# B&R Automation Studio project LiquidControlOfTank
Automation Studio 4.3.7.46 SP

## Configuration Config1

CPU 4PP065.0571-X74, AutomationRuntime E4.34, Build 4.1.2, Vc V4.34.1

### Task classes (Cpu.sw)
```
Cyclic#4:
  Master <- Modbus.Master.prg
  Visu_1 <- Visualisation.Visu_1.prg
DataObjects: datamod <- Modbus.datamod.dob
VcDataObjects: Visu1 <- Visualisation.Visu1.dob
Binaries: udbdef, vcrt, vccnum, vcctext, Visu101, vcpfmtcx, Visu103, Visu102, vcfile, vcgclass, vcpdsw, vccshape, arial, vccbmp, vcmgr, vcchspot, vcdsloc, vcfntttf, vccovl, vcshared, arialbd, vcalarm, vcptelo, vccdt, vccbtn, vcbclass, vcpfpp30, vcdsint, vctcal, TCData, vcpdpp30, vccalarm, vccbar, arconfig, User, ashwd, sysconf, ashwac, Role, asfw, iomap
Libraries: asstring, AsBrStr, DRV_mbus, DataObj, runtime, become, dvframe, vcresman, fileio, asieccon
```

### Hardware
```
4PP065_0571_X74 : 4PP065.0571-X74 v1.1.5.0
  Connector IF5:
    ActivateDevice = 1
    Mode = Manual
    InternetAddress = 192.168.1.10
    SubnetMask = 255.255.255.0
  ConfigurationID = 01082018_Config1
  TimeZone = 260
  VcObjectName = Visu1
4PP065_IF23-1 : 4PP065.IF23-1 v1.0.4.0  [SS -> 4PP065_0571_X74.SS1]
  Connector IF1:
    Baudrate = 19200
    Parity = N
```

## Configuration Config2

CPU X20cCP1301, AutomationRuntime E4.34, Build 4.1.2, Vc V4.34.1

### Task classes (Cpu.sw)
```
Cyclic#4:
  Program1 <- Program1.prg
  Visu_1 <- Visu_1.prg
VcDataObjects: Visu1 <- Visu1.dob
Binaries: vcfile, vcrt, vcfntttf, vcctext, arial, vccdt, vcmgr, vcpkat, vccovl, vccnum, vcpfar00, vcdsint, vcpdvnc, vcshared, Visu102, vcpdsw, vcalarm, vcchspot, vccbtn, Visu101, vcgclass, vcdsloc, arialbd, vcnet, TCData, vctcal, udbdef, Visu103, vcbclass, vccshape, vccbmp, ashwac, User, ashwd, arconfig, sysconf, Role, asfw, iomap
Libraries: become, standard, fileio, dataobj, vcresman, runtime
```

### Hardware
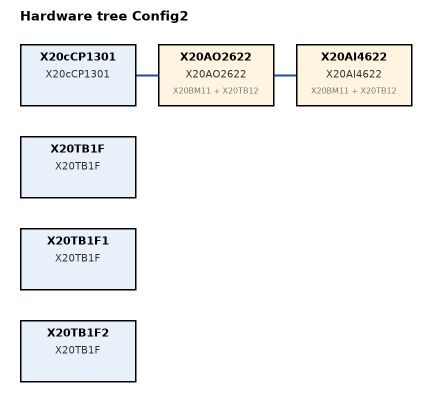
```
X20AI4622 : X20AI4622 v1.0.4.0  [SS1 -> X20TB12a.SS; SL -> X20BM11a.SL1]
  LowerLimit = 0
  ChannelType01 = 4 to 20mA
  ChannelType02 = 4 to 20mA
X20AO2622 : X20AO2622 v1.1.0.0  [SS1 -> X20TB12.SS; SL -> X20BM11.SL1]
  ChannelType01 = 4 to 20mA
  ChannelType02 = 4 to 20mA
X20BM11 : X20BM11 v1.0.0.1  [X2X1 -> X20cCP1301.IF6]
X20BM11a : X20BM11 v1.0.0.1  [X2X1 -> X20BM11.X2X2]
X20TB12 : X20TB12 v1.0.0.0
X20TB12a : X20TB12 v1.0.0.0
X20TB1F : X20TB1F v1.0.0.0
X20TB1F1 : X20TB1F v1.0.0.0
X20TB1F2 : X20TB1F v1.0.0.0
X20cCP1301 : X20cCP1301 v1.3.2.0  [X1 -> X1.SL; X2 -> X2.SL; X3 -> X3.SL]
  Module X1 (Type=X1, Virtual=true, Version=1.3.2.0)
    Connection (Connector=SS1, TargetModule=X20TB1F, TargetConnector=SS)
    Connection (Connector=SL, TargetModule=X20cCP1301, TargetConnector=X1)
  Module X2 (Type=X2, Virtual=true, Version=1.3.2.0)
    Connection (Connector=SS1, TargetModule=X20TB1F1, TargetConnector=SS)
    Connection (Connector=SL, TargetModule=X20cCP1301, TargetConnector=X2)
  Module X3 (Type=X3, Virtual=true, Version=1.3.2.0)
    Connection (Connector=SS1, TargetModule=X20TB1F2, TargetConnector=SS)
    Connection (Connector=SL, TargetModule=X20cCP1301, TargetConnector=X3)
  Connector IF2:
    ActivateDevice = 1
    Mode = Manual
    InternetAddress = 192.168.0.10
    SubnetMask = 255.255.255.0
    Vnc1
    VncVcObjectName1 = Visu1
    VncKeyMappingFile1 = VC\PS2-Keyboard.dis
    VncRefreshRate1 = 100
  ConfigurationID = 01082018_Config2
```

### IoMap.iom - X20cCP1301/IoMap.iom
```iecst
VAR_CONFIG
	::VALVE.feedback.raw AT %IW."X20AI4622".AnalogInput01;
	::TANK.level.raw AT %IW."X20AI4622".AnalogInput02;
	Cyclic#1.::ai_input_status AT %IB."X20AI4622".StatusInput01;
	::PUMP.status_running AT %IX."X2".DigitalInput01;
	::PUMP.status_remote AT %IX."X2".DigitalInput02;
	::VALVE.status_remote AT %IX."X2".DigitalInput03;
	::VALVE.status_local AT %IX."X2".DigitalInput04;
	::VALVE.button_open AT %IX."X2".DigitalInput05;
	::VALVE.button_close AT %IX."X2".DigitalInput06;
	::VALVE.button_stop AT %IX."X2".DigitalInput07;
	::PUMP.cmd_on AT %IX."X3".StatusDigitalOutput01;
	::VALVE.signal_valve_opened AT %IX."X3".StatusDigitalOutput02;
	::VALVE.signal_valve_closed AT %IX."X3".StatusDigitalOutput03;
	::VALVE.cmd_valve_open AT %IX."X3".StatusDigitalOutput04;
	::VALVE.cmd_valve_close AT %IX."X3".StatusDigitalOutput05;
END_VAR
```

## Configuration Config3

CPU X20CP1301, AutomationRuntime E4.34, Build 4.1.2, Vc V4.34.1

### Task classes (Cpu.sw)
```
Cyclic#4:
  Visu_1 <- Visualisation.Visu_1.prg
  Main_Progr <- Main_Program.prg
  Slave <- Modbus.Slave.prg
DataObjects: datamod <- Modbus.datamod.dob
VcDataObjects: Visu1 <- Visualisation.Visu1.dob
Binaries: Visu101, vccbar, vcrt, vcfntttf, vcctext, arial, vccdt, vcmgr, vcpkat, vccovl, vcchspot, vcdsint, vcpfx20, vcpdvnc, vcshared, Visu102, vcpdsw, vcfile, vcalarm, vccbtn, vccnum, vcgclass, vcdsloc, arialbd, vcnet, TCData, vctcal, udbdef, vccalarm, Visu103, vcbclass, vccshape, vccbmp, ashwac, User, ashwd, arconfig, sysconf, Role, asfw, iomap, vcpfar00
Libraries: become, vcresman, fileio, dataobj, ashw, runtime, standard, asstring, drv_mbus, dvframe
```

### Hardware
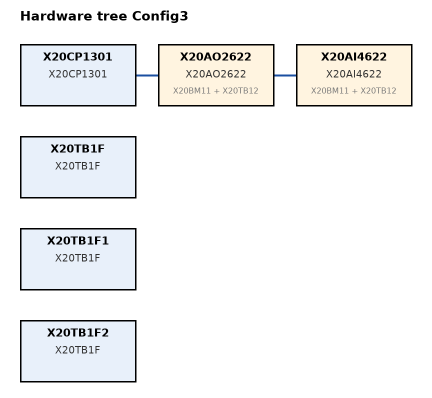
```
X20AI4622 : X20AI4622 v1.0.4.0  [SS1 -> X20TB12.SS; SL -> X20BM11.SL1]
  LowerLimit = 0
  ChannelType01 = 4 to 20mA
  ChannelType02 = 4 to 20mA
  ChannelType03 = 4 to 20mA
  ChannelType04 = 4 to 20mA
X20AO2622 : X20AO2622 v1.1.0.0  [SS1 -> X20TB12a.SS; SL -> X20BM11a.SL1]
  ChannelType01 = 4 to 20mA
  ChannelType02 = 4 to 20mA
X20BM11 : X20BM11 v1.0.0.1  [X2X1 -> X20BM11a.X2X2]
X20BM11a : X20BM11 v1.0.0.1  [X2X1 -> X20CP1301.IF6]
X20CP1301 : X20CP1301 v1.3.2.0  [X1 -> X1.SL; X2 -> X2.SL; X3 -> X3.SL]
  Module X1 (Type=X1, Virtual=true, Version=1.3.2.0)
    Connection (Connector=SS1, TargetModule=X20TB1F, TargetConnector=SS)
    Connection (Connector=SL, TargetModule=X20CP1301, TargetConnector=X1)
  Module X2 (Type=X2, Virtual=true, Version=1.3.2.0)
    Connection (Connector=SS1, TargetModule=X20TB1F1, TargetConnector=SS)
    Connection (Connector=SL, TargetModule=X20CP1301, TargetConnector=X2)
  Module X3 (Type=X3, Virtual=true, Version=1.3.2.0)
    Connection (Connector=SS1, TargetModule=X20TB1F2, TargetConnector=SS)
    Connection (Connector=SL, TargetModule=X20CP1301, TargetConnector=X3)
  Connector IF1:
    Baudrate = 19200
    Parity = N
  Connector IF2:
    ActivateDevice = 1
    Mode = Manual
    InternetAddress = 192.168.1.100
    SubnetMask = 255.255.255.0
    Vnc1
    VncVcObjectName1 = Visu1
    VncKeyMappingFile1 = VC\PS2-Keyboard.dis
    VncRefreshRate1 = 100
  ConfigurationID = LiquidControlOfTank_Config3
X20TB12 : X20TB12 v1.0.0.0
X20TB12a : X20TB12 v1.0.0.0
X20TB1F : X20TB1F v1.0.0.0
X20TB1F1 : X20TB1F v1.0.0.0
X20TB1F2 : X20TB1F v1.0.0.0
```

### IoMap.iom - X20CP1301/IoMap.iom
```iecst
VAR_CONFIG
	::VALVE.feedback.raw AT %IW."X20AI4622".AnalogInput01;
	::TANK.level.raw AT %IW."X20AI4622".AnalogInput02;
	::PUMP.status_running AT %IX."X2".DigitalInput01;
	::PUMP.status_remote AT %IX."X2".DigitalInput02;
	::VALVE.status_remote AT %IX."X2".DigitalInput03;
	::VALVE.status_local AT %IX."X2".DigitalInput04;
	::VALVE.button_open AT %IX."X2".DigitalInput05;
	::VALVE.button_close AT %IX."X2".DigitalInput06;
	::VALVE.button_stop AT %IX."X2".DigitalInput07;
	::PUMP.cmd_on AT %QX."X3".DigitalOutput01;
	::VALVE.signal_valve_opened AT %QX."X3".DigitalOutput02;
	::VALVE.signal_valve_closed AT %QX."X3".DigitalOutput03;
	::VALVE.cmd_valve_open AT %QX."X3".DigitalOutput04;
	::VALVE.cmd_valve_close AT %QX."X3".DigitalOutput05;
END_VAR
```

## Logical view

Binary libraries used (declarations not repeated): operator, runtime, astime, AsIecCon, asstring, AsBrStr, DRV_mbus, DataObj, standard, dvframe

### Global.typ - Global data types
```iecst
TYPE
	Pump_typ : 	STRUCT
		status_running : BOOL; (*Статус насоса "Включен / Выключен"*)
		status_remote : BOOL; (*Статус переключателя "Дистанционный"*)
		cmd_on : BOOL; (*Команда "Включить" насос*)
		button_stop : BOOL; (*Кнопка "Стоп"*)
	END_STRUCT;
	Valve_typ : 	STRUCT
		status_remote : BOOL; (*Статус переключателя "Дистанционный"*)
		status_local : BOOL; (*Статус переключателя "Местный"*)
		button_open : BOOL; (*Кнопка "Открыть" задвижку*)
		button_close : BOOL; (*Кнопка "Закрыть" задвижку*)
		button_stop : BOOL; (*Кнопка "Стоп" задвижку*)
		signal_valve_opened : BOOL; (*Сигнал на индикацию "Задвижка открыта"*)
		signal_valve_closed : BOOL; (*Сигнал на индикацию "Задвижка закрыта"*)
		cmd_valve_open : BOOL; (*Команда открыть задвижку*)
		cmd_valve_close : BOOL; (*Команда закрыть задвижку*)
		feedback : Analog_FB; (*Состояние задвижки (0-100%)*)
	END_STRUCT;
	Tank_typ : 	STRUCT
		level : Analog_FB; (*Уровень жидкости в резервуаре*)
	END_STRUCT;
END_TYPE
```

### Global.var - Global variables
```iecst
(*Задвижка*)
VAR
	VALVE : Valve_typ;
END_VAR
(*Насос*)
VAR
	PUMP : Pump_typ;
END_VAR
(*Резервуар*)
VAR
	TANK : Tank_typ;
END_VAR
(*Аналоговые сигналы*)
VAR
	ai_input_status : USINT; (*Состояние аналоговых каналов*)
END_VAR
(*Примеры для аларма*)
VAR
	alarm : ARRAY[0..19] OF BOOL;
	general_alarm : BOOL;
END_VAR
(*Insert your comment here.*)
VAR
	timer_for_valve : UINT; (*Таймер для открытия задвижки *)
	level_limits : Analog_Limits_typ; (*Технологические значения диапазонов уровня в резервуаре*)
	cmd_pump_on : BOOL; (*Команда для запуска насоса в дистанционном режиме*)
	cmd_pump_off : BOOL; (*Команда для останова насоса в дистанционном режиме*)
	cmd_valve_open : BOOL; (*Команда для открытия задвижки в дистанционном режиме*)
	cmd_valve_close : BOOL; (*Команда для закрытия задвижки в дистанционном режиме*)
	cmd_valve_stop : BOOL; (*Команда для останова задвижки в дистанционном режиме*)
	mode_remote_auto : BOOL; (*Режим дистанционный "Автомат"*)
	mode_remote_manual : BOOL; (*Режим дистанционный "Ручной"*)
	block_auto : BOOL; (*Блокировка кнопки "Автомат" на Touch - панели*)
	block_manual : BOOL; (*Блокировка кнопки "Manual" на Touch - панели*)
	block_valve_cmd : BOOL; (*Блокировка кнопок управления задвижкой в режиме "Дистанционный"*)
	block_pump_cmd : BOOL; (*Блокировка кнопок управления насосом в режиме "Дистанционный"*)
	ack_alarms : BOOL;
END_VAR
```

### Package Logical/Libraries - Global libraries

### Library Logical/Libraries/become (ANSIC, version 1.00.0)

#### Types.typ - Exported data types
```iecst
(*Аналоговый сигнал*)

TYPE
	Analog_Settings_type : 	STRUCT
		scale_h : REAL;
		scale_l : REAL;
		offset : REAL;
	END_STRUCT;
	Analog_Limits_typ : 	STRUCT
		HiHi : REAL;
		Hi : REAL;
		Lo : REAL;
		LoLo : REAL;
		hys : REAL;
	END_STRUCT;
	anaAlarmsEnum :
		(
		SIGNAL_NO_ALARM := 0,
		SIGNAL_OVER := 1,
		SIGNAL_UNDER := 2,
		SIGNAL_OPEN_LINE := 4,
		SIGNAL_HI_HI := 8,
		SIGNAL_HI := 16,
		SIGNAL_LO := 32,
		SIGNAL_LO_LO := 64
		);
END_TYPE

(*Общие*)

TYPE
	localRemoteSwitchEnum :
		( (*Положение ключа управления*)
		SW_OFF := 0,
		SW_LOCAL := 1,
		SW_REMOTE := 2
		);
END_TYPE
```

#### become.fun - Exported functions and function blocks
```iecst
FUNCTION_BLOCK Analog_FB (*Аналоговый сигнал*)
	VAR_INPUT
		raw : INT; (*"сырое" значение с модуля*)
		ai_input_status : BYTE; (*байт-статус с модуля*)
		ai_channel_num : BYTE; (*номер аналогового входа*)
	END_VAR
	VAR_OUTPUT
		value : REAL; (*смасштабированное значение в физических единицах*)
	END_VAR
	VAR
		sett : Analog_Settings_type;
		limits : Analog_Limits_typ;
		alarms : anaAlarmsEnum;
	END_VAR
	VAR_INPUT
		adc_up : INT; (*Верхняя шкала*)
		adc_dn : INT; (*Нижняя шкала*)
	END_VAR
END_FUNCTION_BLOCK
```

#### Analog.c
```c
#include <bur/plctypes.h>
#include "become.h"

void Analog_FB (struct Analog_FB* inst)
{
	INT adc_up = inst->adc_up;
	INT adc_dn = inst->adc_dn;
	REAL raw, phys;
	BOOL signal_fail;
	BYTE status, channel_number;
	anaAlarmsEnum tAlarms = 0;

	/* Диагностика состояния аналогового сигнала*/
	/* Нумерация каналов начинается с 0, поэтому "номер канала" - 1.
	   Статусы каналов разбиты на 2 переменные, поэтому каналы 5-8
	   заново начинаюся с 0, но во второй переменной */

	channel_number = inst->ai_channel_num >4 ? inst->ai_channel_num - 5 : inst->ai_channel_num - 1;

	status = (inst->ai_input_status >> (channel_number << 1)) & 0x03;

	switch (status)
	{
		case 0x01:
			/* Lower limit */
			tAlarms |= SIGNAL_UNDER;
			//raw = inst->sett.scale_l;
			break;
		case 0x02:
			/* Upper limit */
			tAlarms |= SIGNAL_OVER;
			//raw = inst->sett.scale_h;
			break;
		case 0x03:
			/* Обрыв */
			tAlarms |= SIGNAL_OPEN_LINE;
			//raw = inst->sett.scale_l;
			break;
		default:
			//raw = inst->sett.invert_input_scale ? (32767 - inst->raw) : inst->raw;
			raw = inst->raw;
			//tAlarms = signal_no_alarm;
			break;
	}

	signal_fail = (tAlarms != 0);

	/* Представление сигнала в инженерных единицах */
	phys = (raw - adc_dn)*(inst->sett.scale_h - inst->sett.scale_l)/(adc_up - adc_dn) + inst->sett.scale_l + inst->sett.offset;

	inst->alarms = (inst->alarms & ~(SIGNAL_UNDER | SIGNAL_OVER | SIGNAL_OPEN_LINE)) | tAlarms;

	if ((!signal_fail) && (phys >= inst->limits.HiHi))
		inst->alarms |= SIGNAL_HI_HI;
	if ((signal_fail) || (phys < inst->limits.HiHi - inst->limits.hys))
		inst->alarms &= ~SIGNAL_HI_HI;

	if ((!signal_fail) && (phys >= inst->limits.Hi))
		inst->alarms |= SIGNAL_HI;
	if ((signal_fail) || (phys < inst->limits.Hi - inst->limits.hys))
		inst->alarms &= ~SIGNAL_HI;

	if ((!signal_fail) && (phys <= inst->limits.Lo))
		inst->alarms |= SIGNAL_LO;
	if ((signal_fail) || (phys > inst->limits.Lo + inst->limits.hys))
		inst->alarms &= ~SIGNAL_LO;

	if ((!signal_fail) && (phys <= inst->limits.LoLo))
		inst->alarms |= SIGNAL_LO_LO;
	if ((signal_fail) || (phys > inst->limits.LoLo + inst->limits.hys))
		inst->alarms &= ~SIGNAL_LO_LO;

	inst->value = phys;
}
```

### Program Logical/Main_Program (ANSIC)

#### Variables.var
```iecst
VAR
	timer_for_pump : USINT; (*Таймер для запуска насоса*)
	TON_valve : TON; (*Таймер для открытия/закрытия задвижки*)
	TON_pump : TON; (*Таймер для старта/останова насоса*)
	virtual_valve_close : BOOL; (*Самоподхват для кнопки  останова насоса*)
	virtual_valve_open : BOOL; (*Самоподхват для кнопки запуска насоса*)
END_VAR
```

#### Cyclic.c
```c
#include <bur/plc.h>
#include <bur/plctypes.h>
#include <standard.h>
#include <become.h>

#ifdef _DEFAULT_INCLUDES
#include <AsDefault.h>
#endif

_LOCAL BOOL pump_status_changed, pump_prev_status;

/* 	alarm[0] - Авария запуска насоса;
	alarm[1] - Авария открытия задвижки;
	alarm[2] - Авария выключения насоса;
	alarm[3] - Авария закрытия задвижки;
	alarm[4] - Сработала кнопка останова задвижки;
	alarm[5] - Верхний уровень в резервуаре;
	alarm[6] - Нижний уровень в резервуаре;
	alarm[7] - Сработала кнопка останова насоса*/

BOOL TimerValve_func(BOOL start, INT presetTime){

	/* Таймер умножаем на 1000 (равно 1 секунде) */
	TON_valve.IN = start;
	TON_valve.PT = presetTime * 1000;
	TON(&TON_valve);

	return TON_valve.Q;
}

BOOL TimerPump_func(BOOL start, INT presetTime){

	/* Таймер умножаем на 1000 (равно 1 секунде) */
	TON_pump.IN = start;
	TON_pump.PT = presetTime * 1000;
	TON(&TON_pump);

	return TON_pump.Q;
}

void Alarm_func(){

	/* Вержний уровень в резервуаре */
	if (TANK.level.value >= TANK.level.limits.HiHi){
		alarm[5] = 1;
		alarm[6] = 0;
	}
	/* Нижний уровень в резервуаре */
	if(TANK.level.value <= TANK.level.limits.LoLo){
		alarm[6] = 1;
		alarm[5] = 0;
	}
	/* Если уровень в пределах нормы, то сбросить алармы по уровню */
	if ((TANK.level.value > TANK.level.limits.LoLo) && (TANK.level.value < TANK.level.limits.HiHi)){
		alarm[5] = 0;
		alarm[6] = 0;
	}
	if (alarm[0] || alarm[7] || alarm[2]){
		PUMP.cmd_on = 0;
	}
	if (alarm[0]){
		cmd_pump_on = 0;
	}
	if (alarm[2]) {
		cmd_pump_off = 0;
	}
	if (alarm[1] || alarm[4]){
		VALVE.cmd_valve_open = 0;
		cmd_valve_open = 0;
	}
	if (alarm[3] || alarm[4]){
		VALVE.cmd_valve_close = 0;
		cmd_valve_close = 0;
	}
	if (alarm[0] || alarm[1] || alarm[2] || alarm[3]){
		mode_remote_manual = 0;
	}
	if (alarm[0] || alarm[1] || alarm[2] || alarm[3] || alarm[4] || alarm[7]){
		mode_remote_auto = 0;}
}

void _CYCLIC ProgramCyclic(void){

	Alarm_func();
	/* =========================== */
	VALVE.feedback.adc_up = 32767;
	VALVE.feedback.adc_dn = 0;
	Analog_FB(&VALVE.feedback);
	/* =========================== */
	TANK.level.adc_up = 11000;
	TANK.level.adc_dn = 0;
	Analog_FB(&TANK.level);

	/* Мониторинг состояния задвижки */
	VALVE.signal_valve_opened = (VALVE.feedback.value == 100) ? 1 : 0;
	VALVE.signal_valve_closed = (VALVE.feedback.value == 0) ? 1 : 0;

	/* Если насос и задвижка в дистанционном режиме, то разрешение на их запуск с панели" */
	if (PUMP.status_remote || VALVE.status_remote){

		/* При нажатии кнопки "Стоп" запустить триггер */
		if (!VALVE.button_stop){
			mode_remote_auto = 0;
			mode_remote_manual = 0;
			VALVE.cmd_valve_close = 0;
			VALVE.cmd_valve_open = 0;
			cmd_valve_close = 0;
			cmd_valve_open = 0;
			TimerPump_func(0, 0);
			TimerValve_func(0, 0);
			alarm[4] = 1; // Сработала кнопка останова задвижки
		}

		pump_status_changed = PUMP.status_running ^ pump_prev_status;	// Status is changed
		pump_prev_status = PUMP.status_running;						 	// Previous status of pump

		/* При нажатии на кнопку "Стоп" по месту, насос должен остановиться, выйти из всех режимов и обнулить команды */
		if (PUMP.cmd_on && pump_status_changed && (pump_prev_status == 0)){
			PUMP.cmd_on = 0;
			mode_remote_auto = 0;
			mode_remote_manual = 0;
			cmd_pump_on = 0;
			cmd_pump_off = 0;
			alarm[7] = 1;
		}

		/* Если на панели выбран режим "Автомат" */
		if (mode_remote_auto){

			/* Открытие задвижки и включение насоса по достижению верхней уставки */
			if (TANK.level.value >= level_limits.Hi){
				VALVE.cmd_valve_close = 0;
				VALVE.cmd_valve_open = 1;

				/* Если задвижка открылась подаем сигнал на останов насоса */
				if (VALVE.feedback.value == 100){
					TimerValve_func(0, 0);
					VALVE.cmd_valve_open = 0;
					VALVE.signal_valve_opened = 1;
					PUMP.cmd_on = 1;
					alarm[1] = 0;

					/* Насос выключился */
					if (PUMP.status_running){
						TimerPump_func(0, 0);
						alarm[0] = 0;
					}

					/* Если насос не включился */
					if (!PUMP.status_running){
						if (TimerPump_func(1, timer_for_pump)){
							PUMP.cmd_on = 0;
							TimerPump_func(0, 0);
							mode_remote_auto = 0;
							MB0[14] = mode_remote_auto;
							alarm[0] = 1;
						}
					}
				}
				if (VALVE.feedback.value < 100){  /* В течение заданного времени задвижка не открылась*/
					if (TimerValve_func(1, timer_for_valve)){
						VALVE.cmd_valve_open = 0;
						TimerValve_func(0, 0);
						mode_remote_auto = 0;
						MB0[14] = mode_remote_auto;
						alarm[1] = 1;
					}
				}
			}

			/* Закрытие задвижки и выключение насоса по достижению нижней уставки */
			if (TANK.level.value <= level_limits.Lo){
				PUMP.cmd_on = 0;

				/* Насос выключен - сигнал на закрытие задвижки */
				if (!PUMP.status_running){
					VALVE.cmd_valve_open = 0;
					VALVE.cmd_valve_close = 1;
					TimerPump_func(0, 0);
					alarm[2] = 0;

					/* Если задвижка закрылась */
					if (VALVE.feedback.value == 0){
						VALVE.cmd_valve_close = 0;
						VALVE.signal_valve_closed = 1;
						TimerValve_func(0, 0);
						alarm[3] = 0;
					}

					/* Если сработал таймер и задвижка не закрылась */
					if (VALVE.feedback.value > 0){
						if (TimerValve_func(1, timer_for_valve)){
							VALVE.cmd_valve_close = 0;
							VALVE.cmd_valve_open = 0;
							TimerValve_func(0, 0);
							mode_remote_auto = 0;
							MB0[14] = mode_remote_auto;
							alarm[3] = 1;
						}
					}
				}

				/* Если насос не выключился, то-  */
				if (PUMP.status_running){
					if (TimerPump_func(1, timer_for_pump)){
						PUMP.cmd_on = 0;
						TimerPump_func(0, 0);
						mode_remote_auto = 0;
						MB0[14] = mode_remote_auto;
						alarm[2] = 1;
					}
				}
			}
		}

		/* Если на панели выбран режим "Manual" */
		if (mode_remote_manual){

			/* Open valve from Touch panel */
			if (cmd_valve_open){
				VALVE.cmd_valve_close = 0;
				VALVE.cmd_valve_open = 1;

				/* Задаем таймер на открытие задвижки */
				if (VALVE.feedback.value == 100){
					TimerValve_func(0, 0);
					VALVE.cmd_valve_open = 0;
					cmd_valve_open = 0;
					MB0[16] = cmd_valve_open;				// [16] Coil
					VALVE.signal_valve_opened = 1;
					alarm[1] = 0;
				}
				if (VALVE.feedback.value < 100){
					if (TimerValve_func(1, timer_for_valve)){
						VALVE.cmd_valve_open = 0;
						cmd_valve_open = 0;
						MB0[16] = cmd_valve_open;				// [16] Coil
						TimerValve_func(0, 0);
						mode_remote_manual = 0;
						MB0[15] = mode_remote_manual;
						alarm[1] = 1;
					}
				}
			}

			/* Close valve from Touch panel */
			if (cmd_valve_close){
				VALVE.cmd_valve_open = 0;
				VALVE.cmd_valve_close = 1;

				/* Задаем таймер на закрытие задвижки */
				if (VALVE.feedback.value == 0){
					TimerValve_func(0, 0);
					VALVE.cmd_valve_close = 0;
					VALVE.signal_valve_closed = 1;
					cmd_valve_close = 0;
					MB0[17] = cmd_valve_close;				// [17] Coil
					alarm[3] = 0;
				}
				if (VALVE.feedback.value > 0) {
					if(TimerValve_func(1, timer_for_valve)){
						VALVE.cmd_valve_close = 0;
						cmd_valve_close = 0;
						MB0[17] = cmd_valve_close;
						TimerValve_func(0, 0);
						mode_remote_manual = 0;
						MB0[15] = mode_remote_manual;
						alarm[3] = 1;
					}
				}
			}

			/* Turn pump on from Touch panel */
			if (cmd_pump_on){
				PUMP.cmd_on = 1;

				if(PUMP.status_running){
					TimerPump_func(0, 0);
					cmd_pump_on = 0;
					MB0[19] = cmd_pump_on;					// [19] Coil
					alarm[0] = 0;
				}

				/*Если сработал таймер и насос не включился */
				if (!PUMP.status_running){
					if (TimerPump_func(1, timer_for_pump)){
						PUMP.cmd_on = 0;
						cmd_pump_on = 0;
						MB0[19] = cmd_pump_on;					// [19] Coil
						TimerPump_func(0, 0);
						mode_remote_manual = 0;
						MB0[15] = mode_remote_manual;
						alarm[0] = 1;
				}
				}
			}

			/* Turn pump off from Touch panel */
			if (cmd_pump_off){
				PUMP.cmd_on = 0;

				if (!PUMP.status_running){
					TimerPump_func(0, 0);
					cmd_pump_off = 0;
					MB0[20] = cmd_pump_off;					// [20] Coil
					alarm[2] = 0;
				}

				/* Если сработал таймер и насос не выключился (залип пускатель и т.п) */
				if (PUMP.status_running){
					if (TimerPump_func(1, timer_for_pump)){
						PUMP.cmd_on = 0;
						cmd_pump_off = 0;
						MB0[20] = cmd_pump_off;
						TimerPump_func(0, 0);
						mode_remote_manual = 0;
						MB0[15] = mode_remote_manual;
						alarm[2] = 1;
					}
				}
			}

			/* Stop valve from Touch panel */
			if (cmd_valve_stop){
				VALVE.cmd_valve_close = 0;
				VALVE.cmd_valve_open = 0;
				cmd_valve_close = 0;
				cmd_valve_open = 0;
				cmd_valve_stop = 0;
				MB0[18] = cmd_valve_stop;				// [18] Coil
				TimerValve_func (0, 0);
			}
		}
	}

	/* Если переключатель режима насоса не в дистанционном */
	if (!PUMP.status_remote)
		PUMP.cmd_on = 0;

	/* Если переключатель режима задвижки в положении "0" */
	if (!VALVE.status_local && !VALVE.status_remote){
		VALVE.cmd_valve_open = 0;
		VALVE.cmd_valve_close = 0;
		cmd_valve_close = 0;
		cmd_valve_open = 0;
		mode_remote_auto = 0;
		TimerValve_func(0, 0);
		virtual_valve_close = 0;
		virtual_valve_open = 0;
	}

	/* Если переключатель режима задвижки в "Местное"*/
	if (VALVE.status_local){

		//mode_remote_auto = 0;
		//cmd_valve_close = 0;
		//cmd_valve_open = 0;

		/* Если по месту нажаната кнопка "Открыть" */
		if (VALVE.button_open || virtual_valve_open){
			virtual_valve_open = 1;
			VALVE.cmd_valve_close = 0;
			VALVE.cmd_valve_open = 1;

			/* Если сработал таймер и задвижка открылась */
			if (VALVE.feedback.value == 100){
				VALVE.signal_valve_opened = 1;
				VALVE.cmd_valve_open = 0;
				virtual_valve_open = 0;
				TimerValve_func(0, 0);
				alarm[1] = 0;
			}

			 /* В течение заданного времени задвижка не открылась*/
			if (VALVE.feedback.value < 100){
				if (TimerValve_func(1, timer_for_valve)){
					TimerValve_func(0, 0);
					VALVE.cmd_valve_open = 0;
					virtual_valve_open = 0;
					alarm[1] = 1;
				}
			}
		}

		/* Если по месту нажаната кнопка "Закрыть" */
		if (VALVE.button_close || virtual_valve_close){
			virtual_valve_close = 1;
			VALVE.cmd_valve_open = 0;
			VALVE.cmd_valve_close = 1;

			/* Если сработал таймер и задвижка не закрылась */
			if (VALVE.feedback.value == 0){
				VALVE.signal_valve_closed = 1;
				VALVE.cmd_valve_close = 0;
				virtual_valve_close = 0;
				TimerValve_func(0, 0);
				alarm[3] = 0;
			}
			if (TimerValve_func(1, timer_for_valve) && (VALVE.feedback.value > 0)){
				TimerValve_func(0, 0);
				VALVE.cmd_valve_close = 0;
				virtual_valve_close = 0;
				alarm[3] = 1;
			}
		}

		/* Если по месту нажаната кнопка "Стоп" */
		if(!VALVE.button_stop){
			VALVE.cmd_valve_close = 0;
			VALVE.cmd_valve_open = 0;
			TimerPump_func(0,0);
			TimerValve_func(0, 0);
			virtual_valve_close = 0;
			virtual_valve_open = 0;
			alarm[4] = 1; 						// Кнопка "Стоп" по месту
		}

	}
}
```

#### Init.c
```c
#include <bur/plctypes.h>

#ifdef _DEFAULT_INCLUDES
	#include <AsDefault.h>
#endif

void _INIT ProgramInit(void)
{
	VALVE.feedback.sett.scale_h = 100;
	VALVE.feedback.sett.scale_l = 0;
	timer_for_valve = 60;

	TANK.level.sett.scale_h = 0;
	TANK.level.sett.scale_l = 100;

	TANK.level.limits.HiHi = 95;
	TANK.level.limits.Hi = 90;
	TANK.level.limits.Lo = 10;
	TANK.level.limits.LoLo = 5;

	level_limits.Hi = 80;
	level_limits.Lo = 20;
	timer_for_pump = 3;
}
```

- Visualisation Logical/Visualisation (not shown)

### Data object Logical/Modbus/datamod (Simple)

#### datamod.dat
```
"DRVmbus.EventPV4", 03, $01, "DRVmbus.LocalPV4", 0000, 0002
"DRVmbus.EventPV41", 03, $01, "DRVmbus.LocalPV41", 0002, 0009
"DRVmbus.EventPV16", 16, $01, "DRVmbus.LocalPV16", 0002, 0009
"DRVmbus.EventPV1", 01, $01, "DRVmbus.LocalPV1", 0000, 0021
"DRVmbus.EventPV50", 05, $01, "DRVmbus.LocalPV50", 0021, 0001
"DRVmbus.EventPV51", 05, $01, "DRVmbus.LocalPV51", 0022, 0001
"DRVmbus.EventPV52", 05, $01, "DRVmbus.LocalPV52", 0023, 0001
"DRVmbus.EventPV53", 05, $01, "DRVmbus.LocalPV53", 0024, 0001
"DRVmbus.EventPV54", 05, $01, "DRVmbus.LocalPV54", 0025, 0001
"DRVmbus.EventPV55", 05, $01, "DRVmbus.LocalPV55", 0026, 0001
"DRVmbus.EventPV56", 05, $01, "DRVmbus.LocalPV56", 0027, 0001
"DRVmbus.EventPV5",  5, $01,  "DRVmbus.LocalPV5", 0028, 0001

;"LibDRVmbus.EventPV4            ", 16, $01, "LibDRVmbus.LocalPV4            ", 0000, 0003
;"LibDRVmbus.EventPV3            ", 03, $01, "LibDRVmbus.LocalPV3            ", 0000, 0003
; \_____________________________/	|    |    \_____________________________/    |      |
;			 	 |					|    |				  	 |				     |      |
;		   31 Characters		    |    |			   31 Characters  		     |      |_Number of coils or registers
;			 						|    |				   						 |_Offset of the Modbus Variables
;									|    |
;									|    |_Target Address of the slave station
;			 						|
;			 						|_ Modbus function
```

### Types.typ
```iecst
TYPE
	DRVmbus_typ : 	STRUCT
		EventPV1 : BOOL;
		EventPV4 : BOOL;
		EventPV5 : BOOL;
		EventPV41 : BOOL;
		EventPV16 : BOOL;
		EventPV50 : BOOL;
		EventPV51 : BOOL;
		EventPV52 : BOOL;
		EventPV53 : BOOL;
		EventPV54 : BOOL;
		EventPV55 : BOOL;
		EventPV56 : BOOL;
		LocalPV1 : ARRAY[0..27]OF BOOL;
		LocalPV4 : ARRAY[0..10]OF UINT;
		LocalPV5 : BOOL;
		LocalPV41 : ARRAY[0..10]OF UINT;
		LocalPV16 : ARRAY[0..12]OF UINT;
		LocalPV50 : BOOL;
		LocalPV51 : BOOL;
		LocalPV52 : BOOL;
		LocalPV53 : BOOL;
		LocalPV54 : BOOL;
		LocalPV55 : BOOL;
		LocalPV56 : BOOL;
	END_STRUCT;
END_TYPE
```

### Variables.var
```iecst
VAR
	MB4 : ARRAY[0..12] OF UINT;
	MB0 : ARRAY[0..30] OF BOOL;
	DRVmbus : DRVmbus_typ;
END_VAR
```

### Program Logical/Modbus/Master (ANSIC)

#### Main.c - Init, cyclic, exit code
```c
#include <bur/plctypes.h>
#include <string.h>
#include "become.h"

#ifdef _DEFAULT_INCLUDES
	#include <AsDefault.h>
#endif

_LOCAL UDINT ident;
_LOCAL BOOL fMaster, openfailed;
_LOCAL BOOL blockRead, firstInit;
_LOCAL UDINT adr;
_LOCAL USINT i, j;

void _INIT ProgramInit(void)
{
	/* Внутренние переменные для разовой инициализации технологических параметров на панели */
	blockRead = 1;
	firstInit = 1;

	Master.MBMOpen.enable = 1;
	Master.MBMOpen.pDevice = (UDINT) &device;
	Master.MBMOpen.pMode = (UDINT) &mode;
	Master.MBMOpen.pConfig = (UDINT) &config;
	Master.MBMOpen.timeout = 2000;
	Master.MBMOpen.ascii = 0;
	MBMOpen(&Master.MBMOpen);

	if (!Master.MBMOpen.status){
		ident = Master.MBMOpen.ident;
		fMaster = 1;
		openfailed = 0;
	}else{
		fMaster = 0;
		openfailed = 1;
	}
}

void _CYCLIC ProgramCyclic(void)
{
	/* Блокировка кнопок управления задвижкой и насосом, если не выбран режим "Ручной"*/
	if (!mode_remote_manual){
		block_pump_cmd = 1;
		block_valve_cmd = 1;
	}else {
		block_pump_cmd = 0;
		block_valve_cmd = 0;
	}

	/* Если насос и задвижка не в дистанционном режиме, то блокируются кнопки выбора режима "Автомат" либо "Ручное" на Touch-панели */
	if (!PUMP.status_remote || !VALVE.status_remote){
		block_auto = 1;
		//block_manual = 1;
	}else{
		block_auto = 0;
		//block_manual = 0;
	}

	/* Если насос и задвижка в дистанционном режиме, то при нажатии на кнопку "Автомат" на Touch-панели блокируется кнопка "Ручное", и наоборот */
	if (PUMP.status_remote && VALVE.status_remote){
		block_manual = mode_remote_auto ? 1 : 0;
		block_auto = mode_remote_manual ? 1 : 0;
	}

	if (!openfailed && fMaster){
		Master.MBMaster.enable = 1;
		Master.MBMaster.ident = ident;
		MBMaster(&Master.MBMaster);
	}

	DRVmbus.EventPV4 = 1;
	DRVmbus.EventPV1 = 1;

	/* Уровень воды в резервуаре */
	adr = (UDINT) memcpy(&TANK.level.value, &DRVmbus.LocalPV4[0], sizeof(TANK.level.value));						//[0,1] Holding

	/* Запись параметров будет просиходить по нажатию на кнопку */
	if (Cmd_Write){

		/* Задание верхней шкалы*/
		adr = (UDINT) memcpy(&DRVmbus.LocalPV16[0], &TANK.level.sett.scale_h, sizeof(TANK.level.sett.scale_h));	//[2,3] Holding
		/* Задание нижней шкалы*/
		adr = (UDINT) memcpy(&DRVmbus.LocalPV16[2], &TANK.level.sett.scale_l, sizeof(TANK.level.sett.scale_l));	//[4,5] Holding
		/* Задание времени открывания задвижки */
		DRVmbus.LocalPV16[4] = timer_for_valve; 																//[6]   Holding
		/* Задание верхней уставки*/
		adr = (UDINT) memcpy(&DRVmbus.LocalPV16[5], &level_limits.Hi, sizeof(level_limits.Hi));					//[7,8] Holding
		/* Задание нижней уставки*/
		adr = (UDINT) memcpy(&DRVmbus.LocalPV16[7], &level_limits.Lo, sizeof(level_limits.Lo));					//[9,10] Holding

		if(!DRVmbus.EventPV16){
			DRVmbus.EventPV16 = 1;
			Cmd_Write = 0;
		}

	}
	/* Считывание параметров со Slave один раз при запуске панели */
	if (firstInit){

		if (!DRVmbus.EventPV41){

			DRVmbus.EventPV41 = 1;
			//DRVmbus.EventPV41 = 0;
			firstInit = 0;			// Переменная для блокировки считывания параметров только один раз
		}
	}
	else{
		if (!DRVmbus.EventPV41 && blockRead){
			/* Верхняя шкала датчика */
			adr = (UDINT) memcpy(&TANK.level.sett.scale_h, &DRVmbus.LocalPV41[0], sizeof(TANK.level.sett.scale_h));	//[2,3] Holding
			/* Задание нижней шкалы */
			adr = (UDINT) memcpy(&TANK.level.sett.scale_l, &DRVmbus.LocalPV41[2], sizeof(TANK.level.sett.scale_l));	//[4,5] Holding
			/* Задание времени открывания задвижки */
			timer_for_valve = DRVmbus.LocalPV41[4]; 																//[6]   Holding
			/* Задание верхней уставки */
			adr = (UDINT) memcpy(&level_limits.Hi, &DRVmbus.LocalPV41[5], sizeof(level_limits.Hi));					//[7,8] Holding
			/* Задание нижней уставки */
			adr = (UDINT) memcpy(&level_limits.Lo, &DRVmbus.LocalPV41[7], sizeof(level_limits.Lo));					//[9,10] Holding

			blockRead = 0;
		}
	}

	/* Задвижка открыта */
	VALVE.signal_valve_opened = DRVmbus.LocalPV1[0];	// [0] Coil
	/* Задвижка закрыта */
	VALVE.signal_valve_closed = DRVmbus.LocalPV1[1];	// [1] Coil
	/* Задвижка в дистанционном режиме */
	VALVE.status_remote = DRVmbus.LocalPV1[2];			// [2] Coil
	/* Задвижка в местном режиме */
	VALVE.status_local = DRVmbus.LocalPV1[3];			// [3] Coil
	/* Насос в дистанционном режиме */
	PUMP.status_remote = DRVmbus.LocalPV1[4];			// [4] Coil
	/* Насос в работе */
	PUMP.status_running = DRVmbus.LocalPV1[5];			// [5] Coil

	for ( i = 0, j = 6 ; i <= 7; i++){
		alarm[i] = DRVmbus.LocalPV1[j];					// [6] [7] [8] [9] [10] [11] [12] [13] Coils
		j++;
	}

	/* Сброс всех алармов с панели */
	if (ack_alarms){

		if (!DRVmbus.EventPV5){
			DRVmbus.LocalPV5 = ack_alarms;
			DRVmbus.EventPV5 = 1;
			ack_alarms = 0;
		}
	}
	if (DRVmbus.LocalPV5){
		if (!DRVmbus.EventPV5){
			DRVmbus.LocalPV5 = 0;
			DRVmbus.EventPV5 = 1;
		}
	}

	/* Если считываемый сигнал "Режим Автомат" отличается от записываемого*/
	if (DRVmbus.LocalPV1[14] != mode_remote_auto){

		/* Если нет алармов, то разрешение на запись */
		if ((alarm[0] != 1) && (alarm[1] != 1) && (alarm[2] != 1) && (alarm[3] != 1) && (alarm[4] != 1) && (alarm[7] != 1)){
			if (!DRVmbus.EventPV50){
				DRVmbus.LocalPV50 = mode_remote_auto;					// [21] Coil
				DRVmbus.EventPV50 = 1;
			}
		}
		else{
			/* Если есть алармы, то присваиваем счиытваемое значение */
			mode_remote_auto = DRVmbus.LocalPV1[14];		// [14] Coil
			if (!DRVmbus.EventPV50){
				DRVmbus.LocalPV50 = mode_remote_auto;					// [21] Coil
				DRVmbus.EventPV50 = 1;
			}
		}
	}
	if ((DRVmbus.LocalPV1[14] == 0) && (mode_remote_auto == 0)){
		if (!DRVmbus.EventPV50){
			DRVmbus.LocalPV50 = 0;					// [21] Coil
			DRVmbus.EventPV50 = 1;
		}
	}

	/* Если считываемый сигнал "Режим Manual" отличается от записываемого*/
	if (DRVmbus.LocalPV1[15] != mode_remote_manual){

		/* Если нет алармов, то разрешение на запись */
		if ((alarm[0] != 1) && (alarm[1] != 1) && (alarm[2] != 1) && (alarm[3] != 1) && (alarm[4] != 1) && (alarm[7] != 1)){
			if (!DRVmbus.EventPV51){
				DRVmbus.LocalPV51 = mode_remote_manual;					// [22] Coil
				DRVmbus.EventPV51 = 1;
			}
		}
		else{
			if (!DRVmbus.EventPV51){
				mode_remote_manual = DRVmbus.LocalPV1[15];		// [15] Coil
				DRVmbus.LocalPV51 = mode_remote_manual;					// [22] Coil
				DRVmbus.EventPV51 = 1;
			}
		}
	}
	if ((DRVmbus.LocalPV1[15] == 0) && (mode_remote_manual == 0)){
		if (!DRVmbus.EventPV51){
			DRVmbus.LocalPV51 = 0;					// [22] Coil
			DRVmbus.EventPV51 = 1;
		}
	}

	/* Если считываемый сигнал "Openvalve" отличается от записываемого */
	if (DRVmbus.LocalPV1[16] != cmd_valve_open){

		/* Если нет алармов и задвижка не в открытом положении, то разрешение на запись команды открыть задвижку */
		if ((alarm[1] != 1) && (alarm[4] != 1) && !VALVE.signal_valve_opened){
			if (!DRVmbus.EventPV52){
				DRVmbus.LocalPV52 = cmd_valve_open;						// [23] Coil
				DRVmbus.LocalPV53 = 0;
				DRVmbus.EventPV52 = 1;
				DRVmbus.EventPV53 = 1;
			}
		}
		/* Если аларм и задвижка не открыта, либо нет алармов и задвижка открыта, то обнуляем команду */
		if (((alarm[1] || alarm[4]) && !VALVE.signal_valve_opened) || ((alarm[1] != 1) && (alarm[4] != 1) && VALVE.signal_valve_opened)){
			if (!DRVmbus.EventPV52){
				cmd_valve_open = 0;
				DRVmbus.LocalPV52 = cmd_valve_open;						// [23] Coil
				DRVmbus.EventPV52 = 1;
			}
		}
	}

	/* Если считываемый сигнал "Close valve" отличается от записываемого */
	if (DRVmbus.LocalPV1[17] != cmd_valve_close){

		/* Если нет алармов и задвижка не в закрытом положении, то разрешение на запись команды закрыть задвижку */
		if ((alarm[3] != 1) && (alarm[4] != 1) && !VALVE.signal_valve_closed){
			if (!DRVmbus.EventPV53){
				DRVmbus.LocalPV53 = cmd_valve_close;					// [24] Coil
				DRVmbus.LocalPV52 = 0;
				DRVmbus.EventPV53 = 1;
				DRVmbus.EventPV52 = 1;
			}
		}
		/* Если алармы и задвижка не закрыта, либо алармов нет и закрыта задвижка, то следует обнуление команды */
		if (((alarm[3] || alarm[4]) && !VALVE.signal_valve_closed) || ((alarm[3] != 1) && (alarm[4] != 1) && VALVE.signal_valve_closed)){
			if (!DRVmbus.EventPV53){
				cmd_valve_close = 0;
				DRVmbus.LocalPV53 = cmd_valve_close;					// [24] Coil
				DRVmbus.EventPV53 = 1;
			}
		}
	}

	/* Если считываемый сигнал "Stop valve" отличается от записываемого */
	if (cmd_valve_stop){
		if (!DRVmbus.EventPV54 && !DRVmbus.LocalPV54){
			DRVmbus.LocalPV54 = cmd_valve_stop;						// [25] Coil
			DRVmbus.LocalPV52 = 0;
			DRVmbus.LocalPV53 = 0;
			DRVmbus.EventPV54 = 1;
			DRVmbus.EventPV52 = 1;
			DRVmbus.EventPV53 = 1;
			cmd_valve_stop = 0;
			cmd_valve_open = 0;
			cmd_valve_close = 0;
		}
	}
	if (DRVmbus.LocalPV54){
		if (!DRVmbus.EventPV54){

			DRVmbus.LocalPV54 = 0;
			DRVmbus.EventPV54 = 1;
		}
	}

	/* Если считываемый сигнал "Run pump" отличается от записываемого */
	if (DRVmbus.LocalPV1[19] != cmd_pump_on){
		/* Если нет алармов и насос не в работе, то разрешение на запись запуска насоса */
		if ((alarm[0] != 1) && (alarm[7] != 1) && !PUMP.status_running){
			if (!DRVmbus.EventPV55){
				DRVmbus.LocalPV55 = cmd_pump_on;						// [26] Coil
				DRVmbus.EventPV55 = 1;
			}
		}
		/* Если есть аларм и насос не запустился, либо алармов нет и насос запустился, то обнуляем команду */
		if(((alarm[0] || alarm[7]) && !PUMP.status_running) || ((alarm[0] != 1) && (alarm[7] != 1) && PUMP.status_running)){
			if(!DRVmbus.EventPV55){
				cmd_pump_on = 0;
				DRVmbus.LocalPV55 = cmd_pump_on;
				DRVmbus.EventPV55 = 1;
			}
		}
	}

	/* Если считываемый сигнал "остановить насос" отличается от записываемого */
	if (DRVmbus.LocalPV1[20] != cmd_pump_off){
		/* Если нет алармов и насоса в работе, то разрешение на запись останова насоса */
		if ((alarm[2] != 1) && PUMP.status_running){
			if (!DRVmbus.EventPV56){
				DRVmbus.LocalPV56 = cmd_pump_off;						// [27] Coil
				DRVmbus.EventPV56 = 1;
			}
		}
		/* Если есть аларм и насос не выключился, то обнуляем команду */
		if((alarm[2] && PUMP.status_running) || ((alarm[2] == 0) && !PUMP.status_running)){
			if(!DRVmbus.EventPV56){
				cmd_pump_off = 0;
				DRVmbus.LocalPV56 = cmd_pump_off;
				DRVmbus.EventPV56 = 1;
			}
		}
	}
}
void _EXIT ProgramExit(void)
{
	DRVmbus.EventPV1 = 0;
	DRVmbus.EventPV4 = 0;
	DRVmbus.EventPV5 = 0;
	DRVmbus.EventPV16 = 0;
	DRVmbus.EventPV41 = 0;
	DRVmbus.EventPV50 = 0;
	DRVmbus.EventPV51 = 0;
	DRVmbus.EventPV52 = 0;
	DRVmbus.EventPV53 = 0;
	DRVmbus.EventPV54 = 0;
	DRVmbus.EventPV55 = 0;
	DRVmbus.EventPV56 = 0;
}
```

#### Types.typ - Local data types
```iecst
TYPE
	Master_typ : 	STRUCT
		MBMOpen : MBMOpen;
		MBMaster : MBMaster;
		MBMClose : MBMClose;
		MBMCmd : MBMCmd;
		S1 : BOOL; (*command to start sending*)
		S2 : BOOL; (*command to start the MBMClose FUB*)
	END_STRUCT;
END_TYPE
```

#### Variables.var - Local variables
```iecst
VAR
	Master : Master_typ;
	Cmd_Write : BOOL; (*Кнопка записать параметры*)
	mode : STRING[48] := '/PHY=RS232 /PA=N /DB=8 /SB=1 /BD=19200';
	device : STRING[32] := 'SS1.IF1';
	config : STRING[32] := 'datamod';
END_VAR
```

### Program Logical/Modbus/Slave (ANSIC)

#### Types.typ
```iecst
TYPE
	Slave_typ : 	STRUCT
		SOpen01 : MBSOpen;
		Slave01 : MBSlave;
		SClose01 : MBSClose;
	END_STRUCT;
END_TYPE
```

#### Variables.var
```iecst
VAR
	mode : STRING[48];
	device : STRING[32];
	SOpen : MBSOpen;
	Slave : MBSlave;
	SClose : MBSClose;
END_VAR
```

#### Main.c
```c
#include <bur/plctypes.h>
#include <string.h>
#include "become.h"
#include <drv_mbus.h>

#ifdef _DEFAULT_INCLUDES
	#include <AsDefault.h>
#endif

_LOCAL UDINT ident;
_LOCAL BOOL fSlave, openFailed;
_LOCAL UDINT adr;
_LOCAL USINT i, j;

void _INIT ProgramInit(void)
{
	adr = (UDINT) strcpy(device, "IF1");
	adr = (UDINT) strcpy(mode, "/PHY=RS232 /PA=N /DB=8 /SB=1 /BD=19200");

	SOpen.enable = 1;
	SOpen.pDevice = (UDINT) &device;
	SOpen.pMode = (UDINT) &mode;
	SOpen.own_ID = 01;
	SOpen.timeout = 500;
	MBSOpen(&SOpen);

	Slave.ident = SOpen.ident;

	if (!SOpen.status){
		ident = SOpen.ident;
		fSlave = 1;
		openFailed = 0;
	}
	else{
		fSlave = 0;
		openFailed = 1;
	}

	/* Верхняя шкала датчика */
	adr = (UDINT) memcpy (&MB4[2],&TANK.level.sett.scale_h, sizeof(TANK.level.sett.scale_h));	// [2,3]
	/* Нижняя шкала датчика */
	adr = (UDINT) memcpy (&MB4[4],&TANK.level.sett.scale_l, sizeof(TANK.level.sett.scale_l));	// [4,5]
	/* Таймер задвижки */
	MB4[6] = timer_for_valve;																	// [6]
	/* Верхняя уставка */
	adr = (UDINT) memcpy (&MB4[7],&level_limits.Hi, sizeof(level_limits.Hi));					// [7,8]
	/* Нижняя уставка */
	adr = (UDINT) memcpy (&MB4[9],&level_limits.Lo, sizeof(level_limits.Lo));					// [9,10]
}

void _CYCLIC ProgramCyclic(void)
{
	// !openFailed && fSlave
	if (!openFailed && fSlave){

		Slave.enable = 1;
		MBSlave(&Slave);

		/* Уровень воды в резервуаре */
		adr = (UDINT) memcpy (&MB4[0],&TANK.level.value, sizeof(TANK.level.value));                 // [0,1]

		/* Задание верхней шкалы*/
		adr = (UDINT) memcpy (&TANK.level.sett.scale_h, &MB4[2], sizeof(TANK.level.sett.scale_h));	// [2,3]
		/* Задание нижней шкалы*/
		adr = (UDINT) memcpy (&TANK.level.sett.scale_l, &MB4[4], sizeof(TANK.level.sett.scale_l));	// [4,5]
		/* Задание времени открывания задвижки */
		timer_for_valve = MB4[6];																	// [6]
		/* Задание верхней уставки*/
		adr = (UDINT) memcpy (&level_limits.Hi, &MB4[7], sizeof(level_limits.Hi));					// [7,8]
		/* Задание нижней уставки*/
		adr = (UDINT) memcpy (&level_limits.Lo, &MB4[9], sizeof(level_limits.Lo));					// [9,10]

		if (MB0[28]){
			alarm[0] = 0;
			alarm[1] = 0;
			alarm[2] = 0;
			alarm[3] = 0;
			alarm[4] = 0;
			alarm[5] = 0;
			alarm[6] = 0;
			alarm[7] = 0;
		}

		/* Задвижка открыта */
		MB0[0] = VALVE.signal_valve_opened;		// [0] Coil
		/* Задвижка закрыта */
		MB0[1] =  VALVE.signal_valve_closed;	// [1] Coil
		/* Задвижка в дистанционном режиме */
		MB0[2] = VALVE.status_remote;			// [2] Coil
		/* Задвижка в местном режиме */
		MB0[3] = VALVE.status_local;			// [3] Coil
		/* Насос в дистанционном режиме */
		MB0[4] = PUMP.status_remote;			// [4] Coil
		/* Насос в работе */
		MB0[5] = PUMP.status_running;			// [5] Coil

		for ( i = 0, j = 6 ; i <= 7; i++){
			MB0[j] = alarm[i];					// [6] [7] [8] [9] [10] [11] [12] [13] Coils
			j++;
		}

		/* Включить режим "Автомат" */
		mode_remote_auto = MB0[21];				// [21] Coil
		/* Включить режим "Manual" */
		mode_remote_manual = MB0[22];			// [22] Coil
		/* Открытие задвижки */
		cmd_valve_open = MB0[23];				// [23] Coil
		/* Закрытие задвижки */
		cmd_valve_close = MB0[24];				// [24] Coil
		/* Останов задвижки */
		cmd_valve_stop = MB0[25];				// [25] Coil
		/* Запуск насоса */
		cmd_pump_on = MB0[26];					// [26] Coil
		/* Останов насоса */
		cmd_pump_off = MB0[27];					// [27] Coil
	}
}

void _EXIT ProgramExit(void)
{

}
```

Listed in the project but not available here: Logical/Libraries/become/Constants.var
